PROGRAM main
VAR
	Enable AT %QX0.0 : bool;
	DelayTimer : TF_RTO;
	Output AT %QX0.1 : bool;
	ResetTimer AT %QX0.2 : bool;
END_VAR

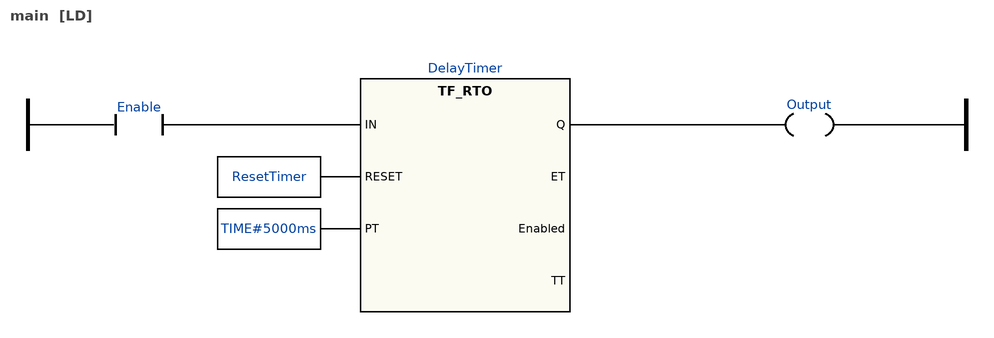
(* LD diagram, written out as Structured Text *)
DelayTimer(IN := Enable, RESET := ResetTimer, PT := TIME#5000ms);
Output := DelayTimer.Q;
END_PROGRAM
